{attribute 'TcGenerated'}
{attribute 'no-analysis'}
{attribute 'linkalways'}
// This function has been automatically generated from the project information.
VAR_GLOBAL CONSTANT
	{attribute 'const_non_replaced'}
	stLibVersion_Actuator : ST_LibVersion := (iMajor := 1, iMinor := 0, iBuild := 0, iRevision := 6, nFlags := 1, sVersion := '1.0.0.6');
END_VAR

(* stored: Version 1.1.0.1, ProductVersion 3.1.4024.12
   GVL Global_Version: Id {b1788d13-8a9c-422f-b449-62f97bbf0a9c} *)
